Universal Robots PolyScope program: TestString.urp

ProgramRoot directory=/home/ur/ursim-3.1/programs; kinematics=(a=[0, -0.612, -0.5723, 0, 0, 0], d=[0.1273, 0, 0, 0.16394, 0.1157, 0.0922], alpha=[1.5708, 0, 0, 1.5708, -1.5708, 0], deltaTheta=[0, 0, 0, 0, 0, 0], status=notInitialized); lastSavedInVersion=(project__name=Polyscope, major__version=3, minor__version=1, svn__revision=16916, build__date=Feb 06 2015, 15:15:00); name=TestString; programVersion=(project__name=PolyScope, major__version=1, minor__version=8, svn__revision=11281, build__date=Aug 07 2013, 11:50:39); robotEnvironmentFileName=default; serialNumberRobot=2014350001
  MainProgram cartesianAcceleration=1.2; cartesianSpeed=0.25; jointAcceleration=1.3962634015954636; jointSpeed=1.0471975511965976; sharedProcessMoveBlendRadius=0.025; motionType=JOINT_SPACE
    Assignment expr="220,150"; operatorValueType=INTEGER; valueSource=EXPRESSION
    Assignment expr="Hello"; operatorValueType=INTEGER; valueSource=EXPRESSION
    Script type=0; expressionBranchNode=StringC = StringA && StringB
    Script type=0; expressionBranchNode=StringC ="[" + StringA + "]"
    Script type=0; expressionBranchNode=popup(StringC)
    Wait 
